// SIMATIC S7-200 project (STEP 7-Micro/WIN), CPU 224 REL 02.01

ORGANIZATION_BLOCK MAIN:OB1
TITLE=PROGRAM COMMENTS
BEGIN
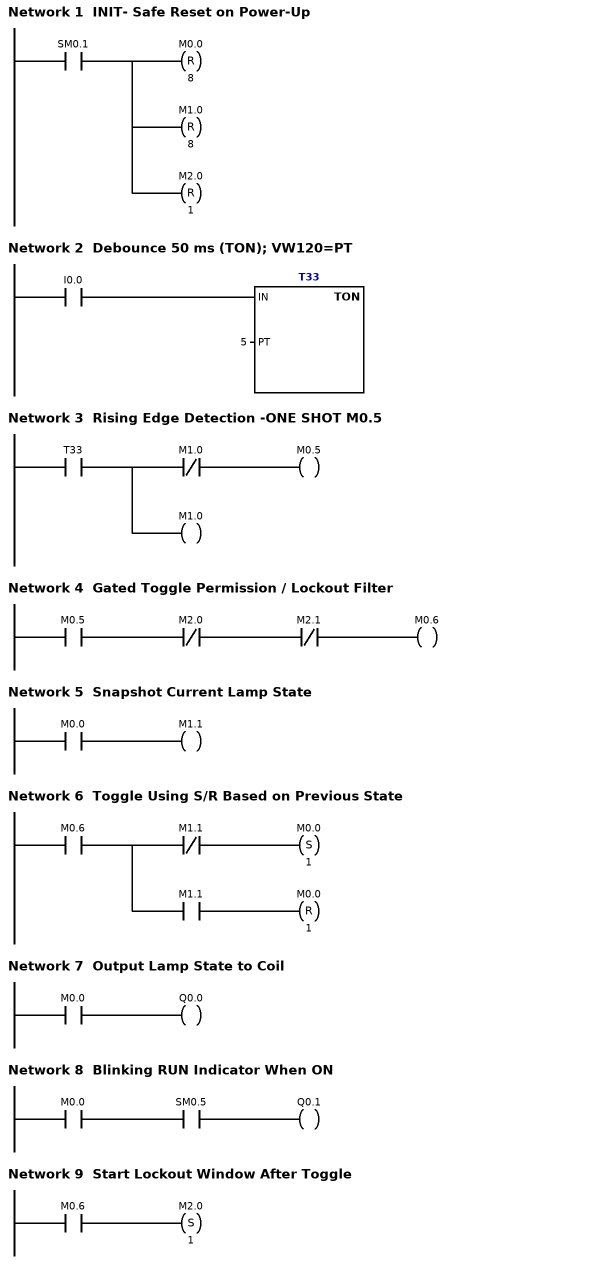
Network 1 // INIT- Safe Reset on Power-Up
LD     SM0.1
R      M0.0, 8
R      M1.0, 8
R      M2.0, 1
Network 2 // Debounce 50 ms (TON); VW120=PT
LD     I0.0
TON    T33, 5
Network 3 // Rising Edge Detection -ONE SHOT M0.5
LD     T33
LPS
AN     M1.0
=      M0.5
LPP
=      M1.0
Network 4 // Gated Toggle Permission / Lockout Filter
LD     M0.5
AN     M2.0
AN     M2.1
=      M0.6
Network 5 // Snapshot Current Lamp State
LD     M0.0
=      M1.1
Network 6 // Toggle Using S/R Based on Previous State
LD     M0.6
LPS
AN     M1.1
S      M0.0, 1
LPP
A      M1.1
R      M0.0, 1
Network 7 // Output Lamp State to Coil
LD     M0.0
=      Q0.0
Network 8 // Blinking RUN Indicator When ON
LD     M0.0
A      SM0.5
=      Q0.1
Network 9 // Start Lockout Window After Toggle
LD     M0.6
S      M2.0, 1
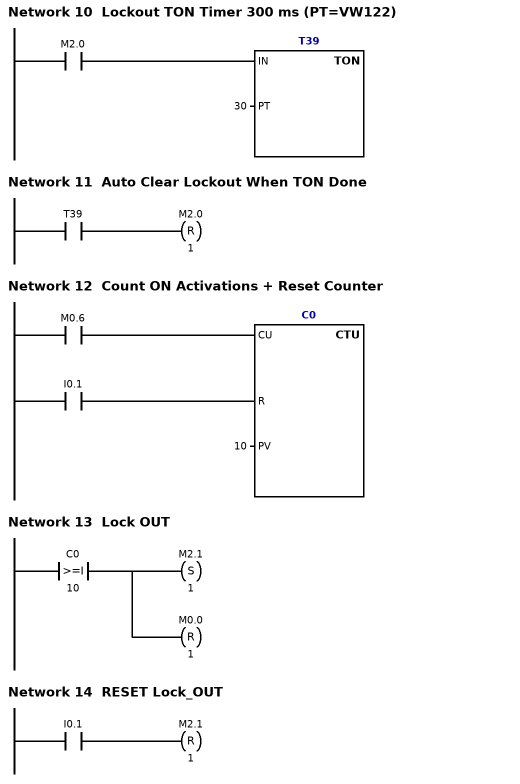
Network 10 // Lockout TON Timer 300 ms (PT=VW122)
LD     M2.0
TON    T39, 30
Network 11 // Auto Clear Lockout When TON Done
LD     T39
R      M2.0, 1
Network 12 // Count ON Activations + Reset Counter
LD     M0.6
LD     I0.1
CTU    C0, 10
Network 13 // Lock OUT
LDW>=  C0, 10
S      M2.1, 1
R      M0.0, 1
Network 14 // RESET Lock_OUT
LD     I0.1
R      M2.1, 1
END_ORGANIZATION_BLOCK
